(*
Nazwa:			P08_CapFeeder
Opis:			Stacja podajnika nasadek
Wersja:			v0.1
Data:			2022-07-13
Autor:			DJ,DP
Urzadzenia:		
Konfiguracja:	
Info:

*)
PROGRAM P08_CapFeeder
VAR_INPUT

END_VAR
VAR
	fbCapFeeder						: FB_CapFeeder;
	fbCapFeederState				: FB_State;	
	eCapFeederState					: E_Station;
	eCapFeederRunningState			: E_CapFeederState; 		// Stan pracy 
	
	IbCapFeederHeightEncoderSetCDone	AT %I*: BOOL;
	IudiCapFeederHeightEncoderCV        AT %I*: UDINT; 
	QbCapFeederHeightEncoderSetC 		AT %Q*: BOOL;		
	QudiCapFeederHeightEncoderSetCV     AT %Q*: UDINT; 	

	QbCapFeederHeightUpCmd 			AT %Q*: BOOL; 					// Wyjście sterujące podnośnikiem podajnika nakrętek, Silnik w górę
	QbCapFeederHeightDownCmd 		AT %Q*: BOOL; 				 	// Wyjście sterujące podnośnikiem podajnika nakrętek, Silnik w dół
	
	QbCapFeederSorterEngine			AT %Q*: BOOL; 					// Wyjście silnikiem sortera
	QbCapFeederSorterAir 			AT %Q*: BOOL; 					// Wyjście sterujące szybkim zaworem wydmuchu
	QbCapFeederSorterAir2 			AT %Q*: BOOL; 					// Wyjście sterujące szybkim zaworem wydmuchu
	
	IbCapFeederSorterCapSensor 		AT %I*: BOOL;					// Wejście z czujnika ultradzwiękowego nasadki sortera
	IbCapFeederFullSleeveSensor		AT %I*: BOOL;					// Wejście przepełnienia rękawa sortera
	IbCapFeederLevelSensor			AT %I*: BOOL;					// Wejście czujnika poziomu sortera

	
	IbFuseCapFeederEngineOK			AT %I*: BOOL;					//Bezpiecznik silnika sortera OK

	IbCapFeederHomingSensor			AT %I*: BOOL;					// Czujnnik bazowania, sorter w gornej pozycji 
	
	QnCapFeederSorterVelocitySV 	AT %Q*: UDINT; 		// Nastawa prędkości
	InCapFeederSorterVelocityCV 	AT %I*: UDINT;		
	InCapFeederSorterSTW 			AT %I*: UINT; 		// Statusword transportera wejściowo wyjściowego
	QnCapFeederSorterCTW 			AT %Q*: UINT;  		// Controlword transportera we/wy
	IbCapFeederSorterWcState		AT %I*: BOOL; 		// Statusword transportera wejściowo wyjściowego

	IbCapFeederPipeSensor			AT %I*: BOOL;		// Czujnik obecnośći flipflopa w rękawie
	
	TimerCapFeederEnable: TOF;
	rtEnable: R_TRIG;
	tonCapFeederEnable: TON;
	
	QbCapFeederGate1 			AT %Q*: BOOL; 					// Wyjście sterujące słabanem #1 w rękawe
	QbCapFeederGate2 			AT %Q*: BOOL; 					// Wyjście sterujące słabanem #1 w rękawe
	
	
	
	bTestW1: BOOL;
END_VAR

aCapFeeder();
aCapFeederWarnings();
QbCapFeederSorterAir2 :=	QbCapFeederSorterEngine OR QbCapFeederSorterAir; //Dodatkowy przedmuch

(* BAZOWANIE - ZMIAN*)
tonCapFeederEnable (IN:=fbCapFeeder.bEnable,PT:=T#5S); (*Dodany ton bo Wizka zjebnie wgrywa zmienne, najpierw włacza Enabla a potem dopiero wybiera recepture*)
rtEnable(CLK:=tonCapFeederEnable.Q,Q=>);
IF rtEnable.Q AND (P00_PackML.fbPMLAuto.ePMLState = E_PMLState.ePMLState_IDLE OR P00_PackML.fbPMLAuto.ePMLState = E_PMLState.ePMLState_EXECUTE)   THEN
		VIS.bCapFeederHeightSet:=TRUE;
ELSIF fbCapFeeder.eState=E_Station.eHomingDone  OR VIS.bErrorOccure THEN
 		VIS.bCapFeederHeightSet:=FALSE;
END_IF
(*KONIEC BAZOWANIE - ZMIANA*)

(*Opoznienie wyłączanie enabla*)
TimerCapFeederEnable(IN:=bCapFeederEnable, PT:=T#2S);

fbCapFeederState(
	eState:=eCapFeederState , 
	bRun:=VIS.bCapFeederRun,	
	eCapFeederRunningState:=eCapFeederRunningState , 
	sStateDesc=> VIS.sCapFeederState,
	iState=>VIS.iCapFeederState	);

ACTION aCapFeeder:
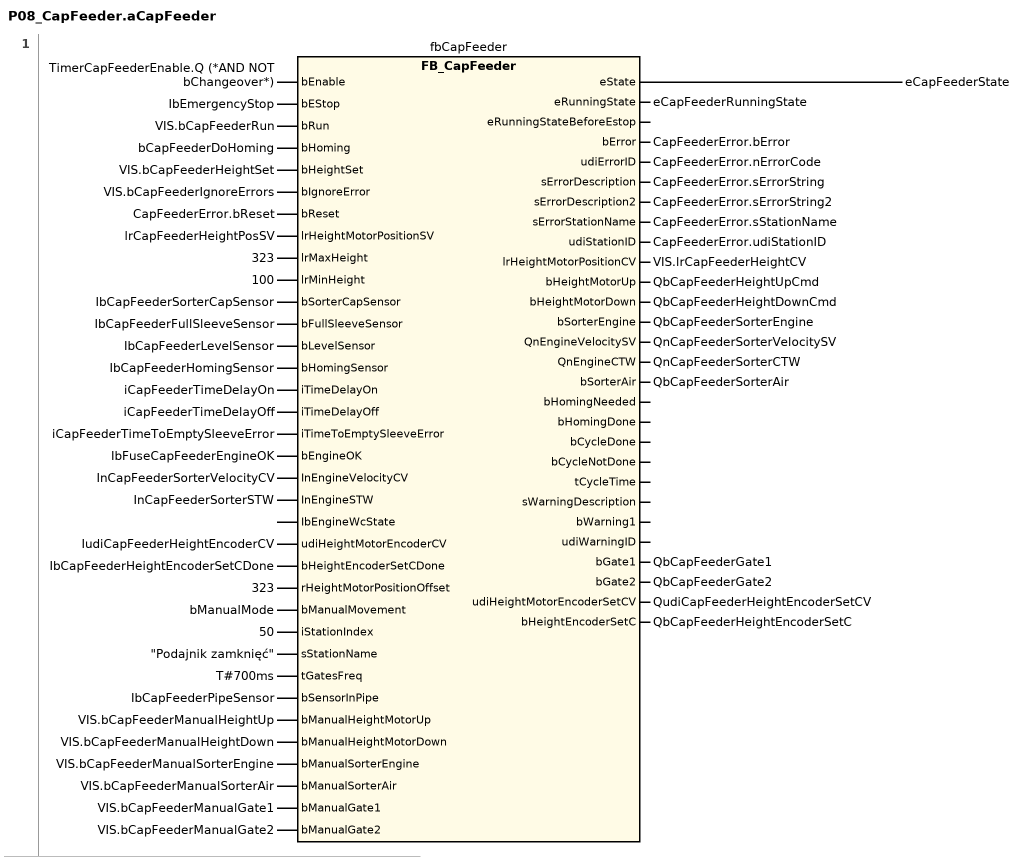
// NETWORK 1
fbCapFeeder(
    bEnable := TimerCapFeederEnable.Q (*AND NOT bChangeover*),
    bEStop := IbEmergencyStop,
    bRun := VIS.bCapFeederRun,
    bHoming := bCapFeederDoHoming,
    bHeightSet := VIS.bCapFeederHeightSet,
    bIgnoreError := VIS.bCapFeederIgnoreErrors,
    bReset := CapFeederError.bReset,
    lrHeightMotorPositionSV := lrCapFeederHeightPosSV,
    lrMaxHeight := 323,
    lrMinHeight := 100,
    bSorterCapSensor := IbCapFeederSorterCapSensor,
    bFullSleeveSensor := IbCapFeederFullSleeveSensor,
    bLevelSensor := IbCapFeederLevelSensor,
    bHomingSensor := IbCapFeederHomingSensor,
    iTimeDelayOn := iCapFeederTimeDelayOn,
    iTimeDelayOff := iCapFeederTimeDelayOff,
    iTimeToEmptySleeveError := iCapFeederTimeToEmptySleeveError,
    bEngineOK := IbFuseCapFeederEngineOK,
    InEngineVelocityCV := InCapFeederSorterVelocityCV,
    InEngineSTW := InCapFeederSorterSTW,
    udiHeightMotorEncoderCV := IudiCapFeederHeightEncoderCV,
    bHeightEncoderSetCDone := IbCapFeederHeightEncoderSetCDone,
    rHeightMotorPositionOffset := 323,
    bManualMovement := bManualMode,
    iStationIndex := 50,
    sStationName := "Podajnik zamknięć",
    tGatesFreq := T#700ms,
    bSensorInPipe := IbCapFeederPipeSensor,
    bManualHeightMotorUp := VIS.bCapFeederManualHeightUp,
    bManualHeightMotorDown := VIS.bCapFeederManualHeightDown,
    bManualSorterEngine := VIS.bCapFeederManualSorterEngine,
    bManualSorterAir := VIS.bCapFeederManualSorterAir,
    bManualGate1 := VIS.bCapFeederManualGate1,
    bManualGate2 := VIS.bCapFeederManualGate2,
    eRunningState => eCapFeederRunningState,
    bError => CapFeederError.bError,
    udiErrorID => CapFeederError.nErrorCode,
    sErrorDescription => CapFeederError.sErrorString,
    sErrorDescription2 => CapFeederError.sErrorString2,
    sErrorStationName => CapFeederError.sStationName,
    udiStationID => CapFeederError.udiStationID,
    lrHeightMotorPositionCV => VIS.lrCapFeederHeightCV,
    bHeightMotorUp => QbCapFeederHeightUpCmd,
    bHeightMotorDown => QbCapFeederHeightDownCmd,
    bSorterEngine => QbCapFeederSorterEngine,
    QnEngineVelocitySV => QnCapFeederSorterVelocitySV,
    QnEngineCTW => QnCapFeederSorterCTW,
    bSorterAir => QbCapFeederSorterAir,
    bGate1 => QbCapFeederGate1,
    bGate2 => QbCapFeederGate2,
    udiHeightMotorEncoderSetCV => QudiCapFeederHeightEncoderSetCV,
    bHeightEncoderSetC => QbCapFeederHeightEncoderSetC); // FB_CapFeeder
eCapFeederState := fbCapFeeder.eState;
END_ACTION

ACTION aCapFeederWarnings:
// Sorter nasadek

IF fbCapFeeder.bWarning1 AND NOT CapFeederWarning[0].bWarning THEN
	CapFeederWarning[0].bWarning										:= TRUE;
	CapFeederWarning[0].udiWarningCode									:= 33;	
	CapFeederWarning[0].sDescription									:= 'Podajnik nasadek | Niski poziom nasadek';
ELSIF NOT fbCapFeeder.bWarning1  AND CapFeederWarning[0].bAcknowledge THEN
	CapFeederWarning[0].bWarning										:= FALSE;
	CapFeederWarning[0].bAcknowledge									:= FALSE;
	VIS.uliWarningAcknowledge.14 										:= FALSE;
ELSIF CapFeederWarning[0].bAcknowledge THEN
	CapFeederWarning[0].bAcknowledge									:= TRUE;
END_IF
END_ACTION

END_PROGRAM

(* stored: Version 1.1.0.1, ProductVersion 3.1.4026.13, FileIdentifier 42acb447447c15d71bc71a2a52f61018853206f6, FileSignature a1b6295366ff74b916d2327c3bd56e405e487ebb0f0a6edca5009bf319e934dfa5620fa9feae8607b9f1845850d3966fcb543f3b16d807bc49b309cee0f5d2d50af7dd212a5a8467dbe4b46bed9c8ab3eda26d293af6a8bca0f9a9a97c1472e43108b6745bef682ab60cde5b857279678387dcc6ccf6087029c8f359d54e2fd6a53f95e5003581f3163534c44f3e0e16c23e17e7c33a2edc01338b085985ca6155e1e463242b575d43913c4019a4402e511c30f99d18b2a88782e2c1b9818103046f7800fd0dc123539a5d57a7fb979bfd631d41393e75248f03a83097204b6e0a83ab9ee899d86607859caa9f5b1ceb7c5d5d061165845a2cf39ca71b20c48f
   POU P08_CapFeeder: Id {98c5bbfe-bd87-4f5f-a215-efdd016278d0}, SpecialFunc None
   Action aCapFeeder: Id {f05bbddc-b67c-4b9c-a02e-0542ec917693}
   Action aCapFeederWarnings: Id {e208a274-4db9-4041-89b1-9a83759dd32e} *)
